{attribute addProperty BoxType "EL5021-0000-0019"}
{attribute addProperty Id "ENC_StatusAT %I*ENC_Status_BA30585080100ENC_ControlAT %Q*ENC_Control_2DBD69A94860WcStateAT %I*WcState_98A4DF7520.250InfoDataAT %I*InfoData_BC63D37F80100"}
{attribute addProperty CRC "3874469664"}
{attribute addProperty SizeInBites "210"}
{attribute addProperty SizeInBytes "26.25"}
TYPE EL5021_1B8188B7 :
STRUCT
	{attribute addProperty Name "ENC_Status"}
	ENC_Status : ENC_Status_BA305850;
	{attribute addProperty Name "ENC_Control"}
	ENC_Control : ENC_Control_2DBD69A9;
	{attribute addProperty Name "WcState"}
	WcState : WcState_98A4DF75;
	{attribute addProperty Name "InfoData"}
	InfoData : InfoData_BC63D37F;
END_STRUCT
END_TYPE

(* stored: Version 1.2.0.0, ProductVersion 3.1.4024.9
   DUT EL5021_1B8188B7: Id {efcd696b-7f29-47df-9d8b-5519de53c8ee} *)
